TYPE ST_ValveScale :
STRUCT
	fPosMax :LREAL := 29490.0;
	fPosMin : LREAL := 20950.0;
	fNegMin : LREAL := 18250.0;
	fNegMax : LREAL := 9830.0;
END_STRUCT
END_TYPE

(* stored: Version 1.1.0.1, ProductVersion 3.1.4024.12
   DUT ST_ValveScale: Id {6320615e-8344-44cb-8d51-3f5a0d70dceb} *)
